TYPE DUT_SetResourcesByName :
STRUCT
	return_value	: DINT;
	ReaourceName	: STRING(50);
	NewData			: STRING(DB.MAX_STRING_SIZE);
END_STRUCT
END_TYPE

(* stored: Version 1.1.0.1, ProductVersion 3.1.4024.15
   DUT DUT_SetResourcesByName: Id {7bfff4b8-45b5-4aea-9a09-8c076b5eb0d0} *)
